SUBAPPLICATION Uebung_002a5_AX (* DigitalInput_I1-3 mit OR auf DigitalOutput_Q1, mit Plug and Socket *)
  (* Standard: 61499-2; Description: Copyright (c) 2023 Meisterschulen am Ostbahnhof This program and the accompanying materials are made available under the terms of the Eclipse Public License 2.0 which is available at https://www.eclipse.org/legal/epl-2.0/ SPDX-License-Identifier: EPL-2.0 *)
  (* Version 1.0, 2023-10-23, Franz Höpfinger, Meisterschulen am Ostbahnhof *)
  IMPORT logiBUS::io::DI::logiBUS_DI::Input_I1;
  IMPORT logiBUS::io::DI::logiBUS_DI::Input_I2;
  IMPORT logiBUS::io::DI::logiBUS_DI::Input_I3;
  IMPORT logiBUS::io::DQ::logiBUS_DO::Output_Q1;
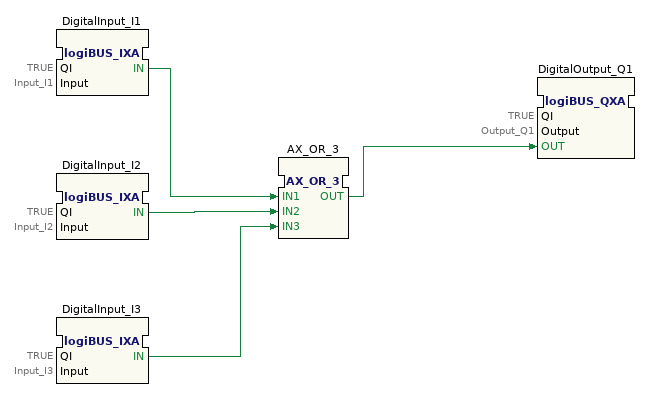
  FBS
    DigitalInput_I1 : logiBUS::io::DI::logiBUS_IXA(QI := TRUE, Input := Input_I1);
    DigitalOutput_Q1 : logiBUS::io::DQ::logiBUS_QXA(QI := TRUE, Output := Output_Q1);
    AX_OR_3 : AX_OR_3;
    DigitalInput_I2 : logiBUS::io::DI::logiBUS_IXA(QI := TRUE, Input := Input_I2);
    DigitalInput_I3 : logiBUS::io::DI::logiBUS_IXA(QI := TRUE, Input := Input_I3);
  END_FBS
  ADAPTER_CONNECTIONS
    AX_OR_3.OUT TO DigitalOutput_Q1.OUT;
    DigitalInput_I1.IN TO AX_OR_3.IN1;
    DigitalInput_I2.IN TO AX_OR_3.IN2;
    DigitalInput_I3.IN TO AX_OR_3.IN3;
  END_CONNECTIONS
END_SUBAPPLICATION
